// SIMATIC S7-200 SMART project (STEP 7-Micro/WIN SMART), CPU SR40

SYMBOL_TABLE 系统符号
Always_On        SM0.0    // 始终接通
First_Scan_On    SM0.1    // 仅在第一个扫描周期时接通
Time_0_Intrvl    SMB34    // 指定中断 0 的时间间隔（从 1 - 255，以 1 ms 递增）。
END_SYMBOL_TABLE

ORGANIZATION_BLOCK MAIN:OB1
TITLE=程序注释
BEGIN
Network 1
// 程序段注释
LD     First_Scan_On:SM0.1
MOVB   0, VB10
MOVB   250, Time_0_Intrvl:SMB34
ATCH   INT_0:INT0, 10
ENI
END_ORGANIZATION_BLOCK

INTERRUPT_BLOCK INT_0:INT0
TITLE=中断例程注释
BEGIN
Network 1
// 程序段注释
LD     Always_On:SM0.0
INCB   VB10
?000
Network 2
LDB=   8, VB10
MOVB   0, VB10
INCB   QB0
?000
END_INTERRUPT_BLOCK
